# EPICS substitutions: app/Db/poe-inj.substitutions
file poeTop.template
{
	{
		FOO = "whatever"
	}
}

file poeChannel.template
{
	pattern
	{ CH }
	{  1 }
	{  2 }
	{  24 }
}
